{attribute 'qualified_only'}
VAR_GLOBAL
END_VAR

(* stored: Version 1.1.0.1, ProductVersion 3.1.4024.12
   GVL GVL_1: Id {fb0ddbc7-c396-49cc-a9ee-dce14b5c7c28} *)
